FUNCTION_BLOCK FB_PulseGenerator
VAR
    PulseOn_TON  : TON;
    PulseOff_TON : TON;
    R_TRIG_0     : R_TRIG;
    Pulse_TON    : TON;
    OutRS        : RS;
    _OnTime      : TIME := T#500MS;
    _OffTime     : TIME := T#500MS;
    _PulseOutput : BOOL;
END_VAR

METHOD CyclicLogic
PulseOn_TON(IN := PulseOutput, PT := _OnTime);
PulseOff_TON(IN := NOT (PulseOutput), PT := _OffTime);
OutRS(SET := PulseOff_TON.Q, RESET1 := PulseOn_TON.Q);
_PulseOutput := OutRS.Q1;
END_METHOD

PROPERTY OffTime : TIME
SET
_OffTime := OffTime;
END_SET
END_PROPERTY

PROPERTY OnTime : TIME
SET
_OnTime := OnTime;
END_SET
END_PROPERTY

PROPERTY PulseOutput : BOOL
GET
PulseOutput := _PulseOutput;
END_GET
END_PROPERTY

END_FUNCTION_BLOCK

(* stored: Version 1.1.0.1
   POU FB_PulseGenerator: Id {2f67ad73-d935-486c-99d8-8cbf25147891}, SpecialFunc None
   Folder I_CyclicFB: Id {eb58122e-03a9-4e13-bcd3-abc3260ce23f}
   Method CyclicLogic: Id {ee5adc93-9924-4c3e-a7be-2748fdab6080}
   Property OffTime: Id {f0bce5f0-e1eb-4294-a906-fdb262faf77f}
   Set Set: Id {6ac0044a-5770-41f9-8b6b-7e3a680f54f3}
   Property OnTime: Id {c67bea88-764c-4168-aecd-4fd7c9ca4d8e}
   Set Set: Id {b5cc1cb7-41f8-4037-ba5d-bfba2fc154cf}
   Property PulseOutput: Id {62e3112e-9d27-41cb-b215-c1827a8e3981}
   Get Get: Id {701e808a-cd3a-40bf-8766-b267ed5bf3f1} *)
